FUNCTION_BLOCK CHECK_TOOL (* Checks if correct tool is attached to the spindle *)
  (* Standard: 61499-2 *)
  (* Version 1.0, 21-03-12, GASR, Universidade do Estado de Santa Catarina *)
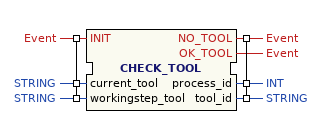
  EVENT_INPUT
    INIT WITH current_tool, workingstep_tool; (* Initialization request *)
  END_EVENT
  EVENT_OUTPUT
    NO_TOOL WITH process_id, tool_id; (* Incorrect tool *)
    OK_TOOL; (* Correct tool *)
  END_EVENT
  VAR_INPUT
    current_tool : STRING; (* Current tool in spindle *)
    workingstep_tool : STRING; (* Tool required *)
  END_VAR
  VAR_OUTPUT
    process_id : INT; (* Process id *)
    tool_id : STRING; (* Tool id *)
  END_VAR
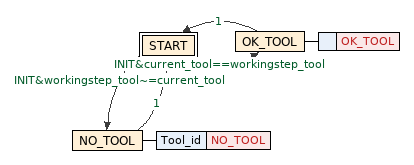
  EC_STATES
    START;
    OK_TOOL : -> OK_TOOL;
    NO_TOOL : Tool_id -> NO_TOOL;
  END_STATES
  EC_TRANSITIONS
    START TO NO_TOOL := INIT&workingstep_tool~=current_tool;
    START TO OK_TOOL := INIT&current_tool==workingstep_tool;
    OK_TOOL TO START := 1;
    NO_TOOL TO START := 1;
  END_TRANSITIONS
  ALGORITHM Tool_id IN Lua:
  process_id = -2  tool_id = workingstep_tool  print( process_id, tool_id )
  END_ALGORITHM
END_FUNCTION_BLOCK
